INTERFACE I_AsyncCommand extends I_Command

METHOD Abort
VAR_INPUT
END_VAR
END_METHOD

PROPERTY PUBLIC Busy : BOOL
GET
END_GET
END_PROPERTY

METHOD PUBLIC CyclicCall
VAR_INPUT
END_VAR
END_METHOD

PROPERTY PUBLIC Done : BOOL
GET
END_GET
END_PROPERTY

PROPERTY PUBLIC Error : BOOL
GET
END_GET
END_PROPERTY

PROPERTY PUBLIC ErrorId : UDINT
GET
END_GET
END_PROPERTY

END_INTERFACE

(* stored: Version 1.1.0.1, ProductVersion 3.1.4024.12
   Itf I_AsyncCommand: Id {1bee37c0-c3a5-0b6f-13cb-01d3f3ae4d04}
   Method Abort: Id {af0faec8-03c9-094f-32c6-8876a661ccc2}
   Property Busy: Id {a78b9e36-0397-00b8-39ab-db80274d7b8a}
   Get Get: Id {07c82fb1-c830-0db9-020e-177357e8ca62}
   Method CyclicCall: Id {33296f58-4355-0dfc-3db1-1173b9e296e6}
   Property Done: Id {0b870abb-a5f7-06bc-24ef-084de0b2b9c7}
   Get Get: Id {f437076f-e9a1-015b-0c19-71fe29723127}
   Property Error: Id {05989871-e6f4-0629-22cf-653120562041}
   Get Get: Id {d3ba6b25-2b2f-03ab-050c-89e678e056e1}
   Property ErrorId: Id {b7cd4ec5-34e3-036b-39ef-cd4663d3b579}
   Get Get: Id {37a6fa1a-e655-0de5-3905-8d5be701e7aa} *)
